// TwinCAT 3 PLC project motor_controller
// ProgramVersion: 3.1.4023.0
// libraries:
//   Tc2_Standard, * (Beckhoff Automation GmbH)
//   Tc2_System, * (Beckhoff Automation GmbH)
//   Tc3_Module, * (Beckhoff Automation GmbH)
// project tree:
//   GVLs/ GVL.TcGVL
//   / PlcTask.TcTTO
//   POUs/ MAIN.TcPOU
// real-time tasks:
//   TASK PlcTask: cycle T#10ms, priority 20, ADS port 350

CONFIGURATION motor_controller
    RESOURCE PLC ON TwinCAT3
        TASK PlcTask(INTERVAL := T#10ms, PRIORITY := 20);
        PROGRAM MAIN WITH PlcTask : MAIN;
    END_RESOURCE
END_CONFIGURATION

// ---- GVLs/GVL.TcGVL
{attribute 'qualified_only'}
VAR_GLOBAL
	
// ***********************************************************************************
// Process inputs
// ***********************************************************************************

// WT ADD 
// Mode 
b_RED_Mode_Manual: BOOL; //Mode
b_RED_Mode_Laptop: BOOL; //Mode


// Temperature and Pressure Sensor
TemperatureAndPressure: STRING := 'TemperatureAndPressure';//***********************************************************
f_RED_Status_Temperature_Funnel_inlet : REAL; // [°C] 
f_RED_Status_Temperature_Funnel_outlet : REAL; // [°C] 
f_RED_Status_Temperature_Funnel_plate : REAL; // [°C] change to concrete pump temperature 

f_RED_Status_Pressure_Funnel_inlet : REAL; // [ bar]

f_RED_Status_Temperature_Concrete_Pump : REAL; // [°C] 
f_RED_Status_Pressure_Concrete_Pump: REAL; // [ bar]

END_VAR

// ---- POUs/MAIN.TcPOU
PROGRAM MAIN
VAR
	Motor_on : BOOL;
	Motor_2_on : BOOL;
END_VAR

END_PROGRAM
